FUNCTION_BLOCK fbMaking_Toast
VAR_INPUT
	CoffeeState : INT;
	BreadInserted : BOOL;
	LeverDown : BOOL;
	Reset : BOOL;
END_VAR
VAR
	step : INT;
	Toasting : BOOL;
	TimerON : TON;
	ToastingDone : BOOL;
END_VAR
VAR_OUTPUT
	MakingToastState : INT;
	ToastWaitTime : BOOL;
	ToastReady : BOOL;
END_VAR

IF Reset THEN
	step := 0;
END_IF
CASE step OF
	0 : //Idle
		ToastingDone := FALSE;
		ToastWaitTime := FALSE;
		LeverDown := FALSE;
		IF BreadInserted AND CoffeeState = 1 THEN
			step := 10;
		END_IF
	10 : // Loading Bread
		IF LeverDown THEN
			Toasting := TRUE;
			ToastWaitTime := TRUE;   // Represent that toast need to wait 5s
			MakingToastState := 1;
		END_IF
		TimerON(IN := Toasting, PT := T#5S);
		ToastingDone := TimerON.Q;
		IF ToastingDone THEN
			ToastReady := TRUE;
			Toasting := FALSE;
			ToastWaitTime := FALSE;   // Reset the representation of waiting
			MakingToastState := 2;
			TimerON(IN := FALSE);
		END_IF
END_CASE

END_FUNCTION_BLOCK

(* stored: Version 1.1.0.1, ProductVersion 3.1.4024.15
   POU fbMaking_Toast: Id {6e6da42b-0686-4a7b-b6de-b1bf9c898711}, SpecialFunc None *)
